// This function has been automatically generated from the project information.
{attribute 'signature_flag' := '1073741824'}
{attribute 'TcGenerated'}
{attribute 'no-analysis'}
FUNCTION F_GetVersion : ST_LibVersion
VAR_INPUT
	
END_VAR

F_GetVersion.iMajor := 1;
F_GetVersion.iMinor := 0;
F_GetVersion.iBuild := 1;
F_GetVersion.iRevision := 0;
F_GetVersion.sVersion := '1.0.1';
F_GetVersion.nFlags := 0;

END_FUNCTION

(* stored: Version 1.1.0.1, ProductVersion 3.1.4024.12
   POU F_GetVersion: Id {00a92cdb-db78-47ba-96a0-d7e7671aca3b}, SpecialFunc None *)
